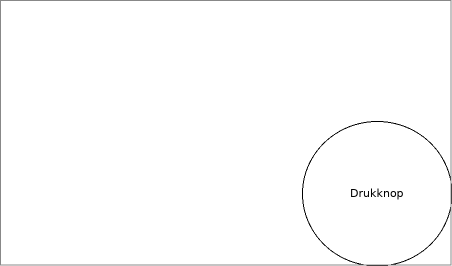
VISUALIZATION Visualization_Click_Logger  // 452x266
    Ellipse (302,121 150x145), "Drukknop"
        tap prg_GetMinimum.bDrukknop
END_VISUALIZATION

(* stored: Version 1.1.0.1, ProductVersion 3.1.4024.15
   Visu Visualization_Click_Logger: Id {7f3a8559-35cc-4971-91a1-9a2b31639110} *)
